KUKA KRL data list: Work_2.dat

&ACCESS RVP
&REL 333
&PARAM EDITMASK = *
&PARAM TEMPLATE = C:\KRC\Roboter\Template\vorgabe
&PARAM DISKPATH = KRC:\R1\Program\HG
DEFDAT  Work_2
;FOLD EXTERNAL DECLARATIONS;%{PE}%MKUKATPBASIS,%CEXT,%VCOMMON,%P
;FOLD BASISTECH EXT;%{PE}%MKUKATPBASIS,%CEXT,%VEXT,%P
EXT  BAS (BAS_COMMAND  :IN,REAL  :IN )
DECL INT SUCCESS
;ENDFOLD (BASISTECH EXT)
;FOLD USER EXT;%{E}%MKUKATPUSER,%CEXT,%VEXT,%P
;Make your modifications here

;ENDFOLD (USER EXT)
;ENDFOLD (EXTERNAL DECLARATIONS)
DECL BASIS_SUGG_T LAST_BASIS={POINT1[] "P0                      ",POINT2[] "P0                      ",CP_PARAMS[] "CPDAT0                  ",PTP_PARAMS[] "PDAT0                   ",CONT[] "                        ",CP_VEL[] "2.0                     ",PTP_VEL[] " 100                    ",SYNC_PARAMS[] "SYNCDAT                 ",SPL_NAME[] "S0                      ",A_PARAMS[] "ADAT0                   "}
DECL E6POS XSURROUND_HOME={X 343.780548,Y 329.155823,Z -382.275,A 0.441927075,B -0.0416149125,C -0.0704164580,S 2,T 10,E1 0.0,E2 0.0,E3 0.0,E4 0.0,E5 0.0,E6 0.0}
DECL FDAT FSurround_Home={TOOL_NO 2,BASE_NO 2,IPO_FRAME #BASE,POINT2[] " ",TQ_STATE FALSE}
DECL PDAT PPDAT1={VEL 100.000,ACC 20.0000,APO_DIST 100.000,GEAR_JERK 50.0000,EXAX_IGN 0}
DECL PDAT PPDAT2={VEL 100.000,ACC 20.0000,APO_DIST 100.000,GEAR_JERK 50.0000,EXAX_IGN 0}
DECL E6POS POS2={X 363.220,Y -0.316000,Z -150.000,A 0.0,B 0.0,C 0.0}
DECL FDAT FS2={TOOL_NO 2,BASE_NO 2,IPO_FRAME #BASE,POINT2[] " ",TQ_STATE FALSE}
DECL LDAT LL2={VEL 0.100000,ACC 100.000,APO_DIST 5.00000,APO_FAC 50.0000,AXIS_VEL 100.000,AXIS_ACC 100.000,ORI_TYP #VAR,CIRC_TYP #BASE,JERK_FAC 50.0000,GEAR_JERK 50.0000,EXAX_IGN 0}
DECL E6POS POS3={X 363.220,Y -0.316000,Z 0.0,A 0.0,B 0.0,C 0.0}
DECL FDAT FS3={TOOL_NO 2,BASE_NO 2,IPO_FRAME #BASE,POINT2[] " ",TQ_STATE FALSE}
DECL LDAT LL3={VEL 0.100000,ACC 100.000,APO_DIST 0.0,APO_FAC 50.0000,AXIS_VEL 100.000,AXIS_ACC 100.000,ORI_TYP #VAR,CIRC_TYP #BASE,JERK_FAC 50.0000,GEAR_JERK 50.0000,EXAX_IGN 0}
DECL E6POS POS4={X 363.395,Y 19.3140,Z 0.0,A 0.0,B 0.0,C 0.0}
DECL FDAT FS4={TOOL_NO 2,BASE_NO 2,IPO_FRAME #BASE,POINT2[] " ",TQ_STATE FALSE}
DECL LDAT LL4={VEL 0.100000,ACC 100.000,APO_DIST 0.0,APO_FAC 50.0000,AXIS_VEL 100.000,AXIS_ACC 100.000,ORI_TYP #VAR,CIRC_TYP #BASE,JERK_FAC 50.0000,GEAR_JERK 50.0000,EXAX_IGN 0}
DECL E6POS POS5={X 363.323059,Y 11.2466183,Z -150.000,A 0.0,B 0.0,C 0.0}
DECL FDAT FS5={TOOL_NO 2,BASE_NO 2,IPO_FRAME #BASE,POINT2[] " ",TQ_STATE FALSE}
DECL LDAT LL5={VEL 0.100000,ACC 100.000,APO_DIST 0.0,APO_FAC 50.0000,AXIS_VEL 100.000,AXIS_ACC 100.000,ORI_TYP #VAR,CIRC_TYP #BASE,JERK_FAC 50.0000,GEAR_JERK 50.0000,EXAX_IGN 0}
DECL E6POS POPM3={X 373.063,Y 22.4860,Z 1.00000,A 0.0,B 0.0,C 0.0}
DECL E6POS POPE3={X 364.614,Y 19.1456451,Z 1.00000,A 0.0,B 0.0,C 20.0000}
DECL FDAT FPE3={TOOL_NO 2,BASE_NO 2,IPO_FRAME #BASE,POINT2[] " ",TQ_STATE FALSE}
DECL LDAT LPM3={VEL 0.01000000,ACC 100.000,APO_DIST 5.00000,APO_FAC 50.0000,AXIS_VEL 100.000,AXIS_ACC 100.000,ORI_TYP #VAR,CIRC_TYP #BASE,JERK_FAC 50.0000,GEAR_JERK 50.0000,EXAX_IGN 0}
DECL E6POS POS6={X 32.5260,Y -0.971000,Z -150.000,A 0.0,B 0.0,C 0.0}
DECL FDAT FS6={TOOL_NO 2,BASE_NO 2,IPO_FRAME #BASE,POINT2[] " ",TQ_STATE FALSE}
DECL LDAT LL6={VEL 0.100000,ACC 100.000,APO_DIST 0.0,APO_FAC 50.0000,AXIS_VEL 100.000,AXIS_ACC 100.000,ORI_TYP #VAR,CIRC_TYP #BASE,JERK_FAC 50.0000,GEAR_JERK 50.0000,EXAX_IGN 0}
DECL E6POS POS7={X 32.5260,Y -0.971000,Z 0.0,A 0.0,B 0.0,C 0.0}
DECL FDAT FS7={TOOL_NO 2,BASE_NO 2,IPO_FRAME #BASE,POINT2[] " ",TQ_STATE FALSE}
DECL LDAT LL7={VEL 0.100000,ACC 100.000,APO_DIST 0.0,APO_FAC 50.0000,AXIS_VEL 100.000,AXIS_ACC 100.000,ORI_TYP #VAR,CIRC_TYP #BASE,JERK_FAC 50.0000,GEAR_JERK 50.0000,EXAX_IGN 0}
DECL E6POS POS8={X 32.3940,Y 18.1940,Z 0.0,A 0.0,B 0.0,C 0.0}
DECL FDAT FS8={TOOL_NO 2,BASE_NO 2,IPO_FRAME #BASE,POINT2[] " ",TQ_STATE FALSE}
DECL LDAT LL8={VEL 0.100000,ACC 100.000,APO_DIST 0.0,APO_FAC 50.0000,AXIS_VEL 100.000,AXIS_ACC 100.000,ORI_TYP #VAR,CIRC_TYP #BASE,JERK_FAC 50.0000,GEAR_JERK 50.0000,EXAX_IGN 0}
DECL E6POS POS9={X 32.4600,Y 8.61150074,Z -150.000,A 0.0,B 0.0,C 0.0}
DECL FDAT FS9={TOOL_NO 2,BASE_NO 2,IPO_FRAME #BASE,POINT2[] " ",TQ_STATE FALSE}
DECL LDAT LL9={VEL 0.100000,ACC 100.000,APO_DIST 0.0,APO_FAC 50.0000,AXIS_VEL 100.000,AXIS_ACC 100.000,ORI_TYP #VAR,CIRC_TYP #BASE,JERK_FAC 50.0000,GEAR_JERK 50.0000,EXAX_IGN 0}
DECL E6POS POPM4={X 22.3930,Y 22.4900,Z 1.00000,A 0.0,B 0.0,C 0.0}
DECL E6POS POPE4={X 20.0512314,Y 30.8929977,Z 0.0,A 0.0,B -20.0000,C 0.0}
DECL FDAT FPE4={TOOL_NO 2,BASE_NO 2,IPO_FRAME #BASE,POINT2[] " ",TQ_STATE FALSE}
DECL LDAT LPM4={VEL 0.0120000,ACC 100.000,APO_DIST 5.00000,APO_FAC 50.0000,AXIS_VEL 100.000,AXIS_ACC 100.000,ORI_TYP #VAR,CIRC_TYP #BASE,JERK_FAC 50.0000,GEAR_JERK 50.0000,EXAX_IGN 0}
DECL E6POS POPM5={X 0.0,Y 0.0,Z 0.0,A 0.0,B 0.0,C 0.0}
DECL E6POS POPE5={X 0.0,Y 0.0,Z 0.0,A 0.0,B 0.0,C 0.0}
DECL FDAT FPE5={TOOL_NO 2,BASE_NO 2,IPO_FRAME #BASE,POINT2[] " ",TQ_STATE FALSE}
DECL LDAT LPM5={VEL 0.0400000,ACC 100.000,APO_DIST 5.00000,APO_FAC 50.0000,AXIS_VEL 100.000,AXIS_ACC 100.000,ORI_TYP #VAR,CIRC_TYP #BASE,JERK_FAC 50.0000,GEAR_JERK 50.0000,EXAX_IGN 0}
DECL E6POS POPM7={X 0.0,Y 0.0,Z 0.0,A 0.0,B 0.0,C 0.0}
DECL E6POS POPE7={X 0.0,Y 0.0,Z 0.0,A 0.0,B 0.0,C 0.0}
DECL FDAT FPE7={TOOL_NO 2,BASE_NO 2,IPO_FRAME #BASE,POINT2[] " ",TQ_STATE FALSE}
DECL LDAT LPM7={VEL 0.0400000,ACC 100.000,APO_DIST 5.00000,APO_FAC 50.0000,AXIS_VEL 100.000,AXIS_ACC 100.000,ORI_TYP #VAR,CIRC_TYP #BASE,JERK_FAC 50.0000,GEAR_JERK 50.0000,EXAX_IGN 0}
DECL E6POS POS10={X 31.6330,Y 679.439,Z -150.000,A 0.0,B 0.0,C 0.0}
DECL FDAT FS10={TOOL_NO 2,BASE_NO 2,IPO_FRAME #BASE,POINT2[] " ",TQ_STATE FALSE}
DECL LDAT LL10={VEL 0.100000,ACC 100.000,APO_DIST 0.0,APO_FAC 50.0000,AXIS_VEL 100.000,AXIS_ACC 100.000,ORI_TYP #VAR,CIRC_TYP #BASE,JERK_FAC 50.0000,GEAR_JERK 50.0000,EXAX_IGN 0}
DECL E6POS POS11={X 31.6330,Y 679.439,Z 0.0,A 0.0,B 0.0,C 0.0}
DECL FDAT FS11={TOOL_NO 2,BASE_NO 2,IPO_FRAME #BASE,POINT2[] " ",TQ_STATE FALSE}
DECL LDAT LL11={VEL 0.100000,ACC 100.000,APO_DIST 0.0,APO_FAC 50.0000,AXIS_VEL 100.000,AXIS_ACC 100.000,ORI_TYP #VAR,CIRC_TYP #BASE,JERK_FAC 50.0000,GEAR_JERK 50.0000,EXAX_IGN 0}
DECL E6POS POS12={X 31.8670,Y 660.025,Z 0.0,A 0.0,B 0.0,C 0.0}
DECL FDAT FS12={TOOL_NO 2,BASE_NO 2,IPO_FRAME #BASE,POINT2[] " ",TQ_STATE FALSE}
DECL LDAT LL12={VEL 0.100000,ACC 100.000,APO_DIST 0.0,APO_FAC 50.0000,AXIS_VEL 100.000,AXIS_ACC 100.000,ORI_TYP #VAR,CIRC_TYP #BASE,JERK_FAC 50.0000,GEAR_JERK 50.0000,EXAX_IGN 0}
DECL E6POS POS13={X 31.7500,Y 669.732056,Z -150.000,A 0.0,B 0.0,C 0.0}
DECL FDAT FS13={TOOL_NO 2,BASE_NO 2,IPO_FRAME #BASE,POINT2[] " ",TQ_STATE FALSE}
DECL LDAT LL13={VEL 0.100000,ACC 100.000,APO_DIST 0.0,APO_FAC 50.0000,AXIS_VEL 100.000,AXIS_ACC 100.000,ORI_TYP #VAR,CIRC_TYP #BASE,JERK_FAC 50.0000,GEAR_JERK 50.0000,EXAX_IGN 0}
DECL E6POS POS14={X 362.986,Y 679.910,Z -150.000,A 0.0,B 0.0,C 0.0}
DECL FDAT FS14={TOOL_NO 2,BASE_NO 2,IPO_FRAME #BASE,POINT2[] " ",TQ_STATE FALSE}
DECL LDAT LL14={VEL 0.100000,ACC 100.000,APO_DIST 0.0,APO_FAC 50.0000,AXIS_VEL 100.000,AXIS_ACC 100.000,ORI_TYP #VAR,CIRC_TYP #BASE,JERK_FAC 50.0000,GEAR_JERK 50.0000,EXAX_IGN 0}
DECL E6POS POS15={X 362.986,Y 679.910,Z 1.00000,A 0.0,B 0.0,C 0.0}
DECL FDAT FS15={TOOL_NO 2,BASE_NO 2,IPO_FRAME #BASE,POINT2[] " ",TQ_STATE FALSE}
DECL LDAT LL15={VEL 0.100000,ACC 100.000,APO_DIST 0.0,APO_FAC 50.0000,AXIS_VEL 100.000,AXIS_ACC 100.000,ORI_TYP #VAR,CIRC_TYP #BASE,JERK_FAC 50.0000,GEAR_JERK 50.0000,EXAX_IGN 0}
DECL E6POS POS16={X 363.044,Y 660.468,Z 1.00000,A 0.0,B 0.0,C 0.0}
DECL FDAT FS16={TOOL_NO 2,BASE_NO 2,IPO_FRAME #BASE,POINT2[] " ",TQ_STATE FALSE}
DECL LDAT LL16={VEL 0.100000,ACC 100.000,APO_DIST 0.0,APO_FAC 50.0000,AXIS_VEL 100.000,AXIS_ACC 100.000,ORI_TYP #VAR,CIRC_TYP #BASE,JERK_FAC 50.0000,GEAR_JERK 50.0000,EXAX_IGN 0}
DECL E6POS POS17={X 363.015,Y 670.188965,Z -150.000,A 0.0,B 0.0,C 0.0}
DECL FDAT FS17={TOOL_NO 2,BASE_NO 2,IPO_FRAME #BASE,POINT2[] " ",TQ_STATE FALSE}
DECL LDAT LL17={VEL 0.100000,ACC 100.000,APO_DIST 0.0,APO_FAC 50.0000,AXIS_VEL 100.000,AXIS_ACC 100.000,ORI_TYP #VAR,CIRC_TYP #BASE,JERK_FAC 50.0000,GEAR_JERK 50.0000,EXAX_IGN 0}
DECL PDAT PPDAT3={VEL 100.000,ACC 20.0000,APO_DIST 100.000,APO_MODE #CDIS,GEAR_JERK 50.0000,EXAX_IGN 0}
DECL FDAT FL0_S2={TOOL_NO 2,BASE_NO 2,IPO_FRAME #BASE,POINT2[] " ",TQ_STATE FALSE}
DECL E6POS POL0_S2={X 0.0,Y 0.0,Z 0.0,A 0.0,B 0.0,C 0.0}
DECL FDAT FL0={TOOL_NO 2,BASE_NO 11,IPO_FRAME #BASE,POINT2[] " ",TQ_STATE FALSE}
DECL E6POS POL0_s4={X 0.0,Y 0.0,Z 0.0,A 0.0,B 0.0,C 0.0}
DECL FDAT FL0_s4={TOOL_NO 2,BASE_NO 2,IPO_FRAME #BASE,POINT2[] " ",TQ_STATE FALSE}
DECL E6POS POC45_S5={X 404.000,Y 36.0000,Z -1.00000,A 0.0,B 20.0000,C 0.0}
DECL FDAT FC45_S5={TOOL_NO 2,BASE_NO 11,IPO_FRAME #BASE,POINT2[] " ",TQ_STATE FALSE}
DECL E6POS POL0_S1={X 376.526398,Y 92.6378174,Z 1.00000,A 0.0,B 20.0000,C 0.0}
DECL FDAT FL0_S1={TOOL_NO 2,BASE_NO 2,IPO_FRAME #BASE,POINT2[] " ",TQ_STATE FALSE}
DECL E6POS POC45_S1={X 376.599762,Y 30.8439941,Z 1.00000,A 0.0,B 20.0000,C 0.0}
DECL FDAT FC45_S1={TOOL_NO 2,BASE_NO 2,IPO_FRAME #BASE,POINT2[] " ",TQ_STATE FALSE}
DECL LDAT LL0_L1={VEL 0.200000,ACC 50.0000,APO_DIST 5.00000,APO_FAC 50.0000,AXIS_VEL 100.000,AXIS_ACC 100.000,ORI_TYP #VAR,CIRC_TYP #BASE,JERK_FAC 50.0000,GEAR_JERK 50.0000,EXAX_IGN 0}
DECL LDAT LC45_L1={VEL 0.0250000,ACC 100.000,APO_DIST 5.00000,APO_FAC 50.0000,AXIS_VEL 100.000,AXIS_ACC 100.000,ORI_TYP #VAR,CIRC_TYP #BASE,JERK_FAC 50.0000,GEAR_JERK 50.0000,EXAX_IGN 0}
DECL E6POS POL90_S1={X 331.308502,Y 19.0502167,Z 1.00000,A 0.0,B 0.0,C 20.0000}
DECL FDAT FL90_S1={TOOL_NO 2,BASE_NO 2,IPO_FRAME #BASE,POINT2[] " ",TQ_STATE FALSE}
DECL LDAT LL90_L1={VEL 0.0250000,ACC 100.000,APO_DIST 5.00000,APO_FAC 50.0000,AXIS_VEL 100.000,AXIS_ACC 100.000,ORI_TYP #VAR,CIRC_TYP #BASE,JERK_FAC 50.0000,GEAR_JERK 50.0000,EXAX_IGN 0}
DECL E6POS POL90_S2={X 198.086502,Y 19.0685,Z 1.00000,A 0.0,B 0.0,C 20.0000}
DECL FDAT FL90_S2={TOOL_NO 2,BASE_NO 2,IPO_FRAME #BASE,POINT2[] " ",TQ_STATE FALSE}
DECL LDAT LL90_L2={VEL 0.0250000,ACC 100.000,APO_DIST 5.00000,APO_FAC 50.0000,AXIS_VEL 100.000,AXIS_ACC 100.000,ORI_TYP #VAR,CIRC_TYP #BASE,JERK_FAC 50.0000,GEAR_JERK 50.0000,EXAX_IGN 0}
DECL E6POS POL90_S3={X 64.8645,Y 19.0867844,Z 1.00000,A 0.0,B 0.0,C 20.0000}
DECL FDAT FL90_S3={TOOL_NO 2,BASE_NO 2,IPO_FRAME #BASE,POINT2[] " ",TQ_STATE FALSE}
DECL LDAT LL90_L3={VEL 0.0250000,ACC 100.000,APO_DIST 5.00000,APO_FAC 50.0000,AXIS_VEL 100.000,AXIS_ACC 100.000,ORI_TYP #VAR,CIRC_TYP #BASE,JERK_FAC 50.0000,GEAR_JERK 50.0000,EXAX_IGN 0}
DECL E6POS POC135_S1={X 31.5589905,Y 18.8913536,Z 1.00000,A 0.0,B 0.0,C 20.0000}
DECL FDAT FC135_S1={TOOL_NO 2,BASE_NO 2,IPO_FRAME #BASE,POINT2[] " ",TQ_STATE FALSE}
DECL LDAT LC135_L1={VEL 0.0250000,ACC 100.000,APO_DIST 5.00000,APO_FAC 50.0000,AXIS_VEL 100.000,AXIS_ACC 100.000,ORI_TYP #VAR,CIRC_TYP #BASE,JERK_FAC 50.0000,GEAR_JERK 50.0000,EXAX_IGN 0}
DECL E6POS POL180_S1={X 0.0,Y 0.0,Z 0.0,A 0.0,B 0.0,C 0.0}
DECL FDAT FL180_S1={TOOL_NO 2,BASE_NO 2,IPO_FRAME #BASE,POINT2[] " ",TQ_STATE FALSE}
DECL LDAT LL180_L1={VEL 0.0400000,ACC 100.000,APO_DIST 0.0,APO_FAC 50.0000,AXIS_VEL 100.000,AXIS_ACC 100.000,ORI_TYP #VAR,CIRC_TYP #BASE,JERK_FAC 50.0000,GEAR_JERK 50.0000,EXAX_IGN 0}
DECL E6POS POL180_S2={X 0.0,Y 0.0,Z 0.0,A 0.0,B 0.0,C 0.0}
DECL FDAT FL180_S2={TOOL_NO 2,BASE_NO 2,IPO_FRAME #BASE,POINT2[] " ",TQ_STATE FALSE}
DECL LDAT LL180_L2={VEL 0.0400000,ACC 100.000,APO_DIST 0.0,APO_FAC 50.0000,AXIS_VEL 100.000,AXIS_ACC 100.000,ORI_TYP #VAR,CIRC_TYP #BASE,JERK_FAC 50.0000,GEAR_JERK 50.0000,EXAX_IGN 0}
DECL E6POS POL180_S3={X 0.0,Y 0.0,Z 0.0,A 0.0,B 0.0,C 0.0}
DECL FDAT FL180_S3={TOOL_NO 2,BASE_NO 2,IPO_FRAME #BASE,POINT2[] " ",TQ_STATE FALSE}
DECL LDAT LL180_L3={VEL 0.0400000,ACC 100.000,APO_DIST 0.0,APO_FAC 50.0000,AXIS_VEL 100.000,AXIS_ACC 100.000,ORI_TYP #VAR,CIRC_TYP #BASE,JERK_FAC 50.0000,GEAR_JERK 50.0000,EXAX_IGN 0}
DECL E6POS POC225_S1={X 0.0,Y 0.0,Z 0.0,A 0.0,B 0.0,C 0.0}
DECL FDAT FC225_S1={TOOL_NO 2,BASE_NO 2,IPO_FRAME #BASE,POINT2[] " ",TQ_STATE FALSE}
DECL LDAT LC225_L1={VEL 0.0400000,ACC 100.000,APO_DIST 0.0,APO_FAC 50.0000,AXIS_VEL 100.000,AXIS_ACC 100.000,ORI_TYP #VAR,CIRC_TYP #BASE,JERK_FAC 50.0000,GEAR_JERK 50.0000,EXAX_IGN 0}
DECL E6POS POL270_S1={X 0.0,Y 0.0,Z 0.0,A 0.0,B 0.0,C 0.0}
DECL FDAT FL270_S1={TOOL_NO 2,BASE_NO 2,IPO_FRAME #BASE,POINT2[] " ",TQ_STATE FALSE}
DECL LDAT Ll270_L1={VEL 0.0400000,ACC 100.000,APO_DIST 0.0,APO_FAC 50.0000,AXIS_VEL 100.000,AXIS_ACC 100.000,ORI_TYP #VAR,CIRC_TYP #BASE,JERK_FAC 50.0000,GEAR_JERK 50.0000,EXAX_IGN 0}
DECL E6POS POL270_S2={X 0.0,Y 0.0,Z 0.0,A 0.0,B 0.0,C 0.0}
DECL FDAT FL270_S2={TOOL_NO 2,BASE_NO 2,IPO_FRAME #BASE,POINT2[] " ",TQ_STATE FALSE}
DECL LDAT LL270_L2={VEL 0.0400000,ACC 100.000,APO_DIST 0.0,APO_FAC 50.0000,AXIS_VEL 100.000,AXIS_ACC 100.000,ORI_TYP #VAR,CIRC_TYP #BASE,JERK_FAC 50.0000,GEAR_JERK 50.0000,EXAX_IGN 0}
DECL E6POS POL270_S3={X 0.0,Y 0.0,Z 0.0,A 0.0,B 0.0,C 0.0}
DECL FDAT FL270_S3={TOOL_NO 2,BASE_NO 2,IPO_FRAME #BASE,POINT2[] " ",TQ_STATE FALSE}
DECL LDAT LL270_L3={VEL 0.0400000,ACC 100.000,APO_DIST 0.0,APO_FAC 50.0000,AXIS_VEL 100.000,AXIS_ACC 100.000,ORI_TYP #VAR,CIRC_TYP #BASE,JERK_FAC 50.0000,GEAR_JERK 50.0000,EXAX_IGN 0}
DECL E6POS POC315_S1={X 0.0,Y 0.0,Z 0.0,A 0.0,B 0.0,C 0.0}
DECL FDAT FC315_S1={TOOL_NO 2,BASE_NO 2,IPO_FRAME #BASE,POINT2[] " ",TQ_STATE FALSE}
DECL LDAT LC315_L1={VEL 0.0400000,ACC 100.000,APO_DIST 0.0,APO_FAC 50.0000,AXIS_VEL 100.000,AXIS_ACC 100.000,ORI_TYP #VAR,CIRC_TYP #BASE,JERK_FAC 50.0000,GEAR_JERK 50.0000,EXAX_IGN 0}
DECL LDAT LL0_L2={VEL 0.0400000,ACC 100.000,APO_DIST 0.0,APO_FAC 50.0000,AXIS_VEL 100.000,AXIS_ACC 100.000,ORI_TYP #VAR,CIRC_TYP #BASE,JERK_FAC 50.0000,GEAR_JERK 50.0000,EXAX_IGN 0}
DECL E6POS POL0_S3={X 0.0,Y 0.0,Z 0.0,A 0.0,B 0.0,C 0.0}
DECL FDAT FL0_S3={TOOL_NO 2,BASE_NO 2,IPO_FRAME #BASE,POINT2[] " ",TQ_STATE FALSE}
DECL LDAT LL0_L3={VEL 0.0400000,ACC 100.000,APO_DIST 0.0,APO_FAC 50.0000,AXIS_VEL 100.000,AXIS_ACC 100.000,ORI_TYP #VAR,CIRC_TYP #BASE,JERK_FAC 50.0000,GEAR_JERK 50.0000,EXAX_IGN 0}
DECL LDAT LL0_L4={VEL 0.0400000,ACC 100.000,APO_DIST 0.0,APO_FAC 50.0000,AXIS_VEL 100.000,AXIS_ACC 100.000,ORI_TYP #VAR,CIRC_TYP #BASE,JERK_FAC 50.0000,GEAR_JERK 50.0000,EXAX_IGN 0}
DECL E6POS XP2={X 293.122131,Y 89.9176636,Z -80.0293961,A 0.441927075,B -0.0416149199,C -0.0704164207,S 2,T 10,E1 0.0,E2 0.0,E3 0.0,E4 0.0,E5 0.0,E6 0.0}
DECL FDAT Fp2={TOOL_NO 2,BASE_NO 2,IPO_FRAME #BASE,POINT2[] " ",TQ_STATE FALSE}
DECL LDAT LCPDAT1={VEL 2.00000,ACC 100.000,APO_DIST 100.000,APO_FAC 50.0000,AXIS_VEL 100.000,AXIS_ACC 100.000,ORI_TYP #VAR,CIRC_TYP #BASE,JERK_FAC 50.0000,GEAR_JERK 50.0000,EXAX_IGN 0}
DECL E6POS XP3={X -42.3839874,Y 91.8151550,Z -80.0254822,A 0.441927075,B -0.0416149236,C -0.0704165,S 2,T 10,E1 0.0,E2 0.0,E3 0.0,E4 0.0,E5 0.0,E6 0.0}
DECL FDAT Fp3={TOOL_NO 2,BASE_NO 2,IPO_FRAME #BASE,POINT2[] " ",TQ_STATE FALSE}
DECL LDAT LCPDAT2={VEL 2.00000,ACC 100.000,APO_DIST 100.000,APO_FAC 50.0000,AXIS_VEL 100.000,AXIS_ACC 100.000,ORI_TYP #VAR,CIRC_TYP #BASE,JERK_FAC 50.0000,GEAR_JERK 50.0000,EXAX_IGN 0}
DECL E6POS XP4={X -39.7999954,Y 716.082336,Z -80.0293350,A 0.441927075,B -0.0416149311,C -0.0704164803,S 2,T 10,E1 0.0,E2 0.0,E3 0.0,E4 0.0,E5 0.0,E6 0.0}
DECL FDAT Fp4={TOOL_NO 2,BASE_NO 2,IPO_FRAME #BASE,POINT2[] " ",TQ_STATE FALSE}
DECL LDAT LCPDAT3={VEL 2.00000,ACC 100.000,APO_DIST 100.000,APO_FAC 50.0000,AXIS_VEL 100.000,AXIS_ACC 100.000,ORI_TYP #VAR,CIRC_TYP #BASE,JERK_FAC 50.0000,GEAR_JERK 50.0000,EXAX_IGN 0}
DECL E6POS XP5={X 294.984924,Y 714.198059,Z -80.0293350,A 0.441927075,B -0.0416149311,C -0.0704164803,S 2,T 10,E1 0.0,E2 0.0,E3 0.0,E4 0.0,E5 0.0,E6 0.0}
DECL FDAT Fp5={TOOL_NO 2,BASE_NO 2,IPO_FRAME #BASE,POINT2[] " ",TQ_STATE FALSE}
DECL LDAT LCPDAT4={VEL 2.00000,ACC 100.000,APO_DIST 100.000,APO_FAC 50.0000,AXIS_VEL 100.000,AXIS_ACC 100.000,ORI_TYP #VAR,CIRC_TYP #BASE,JERK_FAC 50.0000,GEAR_JERK 50.0000,EXAX_IGN 0}
DECL PDAT PPDAT4={VEL 100.000,ACC 20.0000,APO_DIST 100.000,GEAR_JERK 50.0000,EXAX_IGN 0}
ENDDAT
